FUNCTION "FC_SimNoria" : Void
{ S7_Optimized_Access := 'TRUE' }
VERSION : 2.2
// ==============================================================================
// FC_SimNoria - Симулятор фізики та несправностей норії
// ==============================================================================
// Версія: 2.2.0
// Дата: 2026-04-10
// ==============================================================================
// Зміни v2.2:
//   - Видалено симуляцію DI_Feedback_OK та SimFault_Feedback
//   - Видалено параметри SimFault_Feedback та FaultTime_Feedback_ms
//   - Оновлено симуляцію Noria для Breaker/Alignment
//   - Видалено Feedback_Tripped із внутрішнього стану
// ==============================================================================
// Комунікація з FC_Noria ТІЛЬКИ через сигнали:
//   - Читає:  DB_Mechs.Noria[NoriaIdx].DO_Run
//   - Пише:   DB_Mechs.Noria[NoriaIdx].DI_Speed_OK
//             DB_Mechs.Noria[NoriaIdx].DI_Breaker_OK
//             DB_Mechs.Noria[NoriaIdx].DI_Alingment_OK
// ==============================================================================
   VAR_INPUT
      NoriaIdx : Int;
      StartupTime_ms : DInt;
      StopTime_ms : DInt;
      SimFault_Breaker : Bool;
      FaultTime_Breaker_ms : DInt;
      SimFault_Alignment : Bool;
      FaultTime_Alignment_ms : DInt;
      ManualReset : Bool;
   END_VAR

   VAR_TEMP
      idx : Int;
      elapsedMs : DInt;
      nowTck : DInt;
      startupTimeout : Bool;
      stopTimeout : Bool;
      breakerTimeout : Bool;
      alignmentTimeout : Bool;
   END_VAR


BEGIN
    // =========================================================
    // VALIDATE INDEX
    // =========================================================
    IF #NoriaIdx >= 32 THEN
        RETURN;
    END_IF;

    #idx := #NoriaIdx;

    // =========================================================
    // PHASE 0: Ручний скид аварій
    // =========================================================
    IF #ManualReset THEN
        "DB_SimMechs".Noria[#idx].Breaker_Tripped := FALSE;
        "DB_SimMechs".Noria[#idx].Alignment_Tripped := FALSE;
    END_IF;

    // =========================================================
    // PHASE 1: Edge detection DO_Run
    // =========================================================
    IF "DB_Mechs".Noria[#idx].DO_Run AND NOT "DB_SimMechs".Noria[#idx].LastDO_Run THEN
        "DB_SimMechs".Noria[#idx].MotorStartTck := TIME_TCK();
        "DB_SimMechs".Noria[#idx].FaultStartTck := TIME_TCK();
        "DB_SimMechs".Noria[#idx].IsMotorRunning := TRUE;
        "DB_SimMechs".Noria[#idx].IsSpinningUp := TRUE;
        "DB_SimMechs".Noria[#idx].IsSpinningDown := FALSE;
    END_IF;

    IF NOT "DB_Mechs".Noria[#idx].DO_Run AND "DB_SimMechs".Noria[#idx].LastDO_Run THEN
        "DB_SimMechs".Noria[#idx].MotorStopTck := TIME_TCK();
        "DB_SimMechs".Noria[#idx].IsMotorRunning := FALSE;
        "DB_SimMechs".Noria[#idx].IsSpinningUp := FALSE;
        "DB_SimMechs".Noria[#idx].IsSpinningDown := TRUE;
    END_IF;

    "DB_SimMechs".Noria[#idx].LastDO_Run := "DB_Mechs".Noria[#idx].DO_Run;

    // =========================================================
    // PHASE 2: Симуляція DI_Speed_OK (тахо)
    // =========================================================
    IF "DB_SimMechs".Noria[#idx].IsSpinningUp THEN
        #startupTimeout := "FC_TimeElapsedMs"(
                                              StartTck := "DB_SimMechs".Noria[#idx].MotorStartTck,
                                              TimeoutMs := #StartupTime_ms,
                                              ElapsedMs => #elapsedMs,
                                              NowTck => #nowTck
        );
        IF #startupTimeout THEN
            "DB_Mechs".Noria[#idx].DI_Speed_OK := TRUE;
            "DB_SimMechs".Noria[#idx].IsSpinningUp := FALSE;
        ELSE
            "DB_Mechs".Noria[#idx].DI_Speed_OK := FALSE;
        END_IF;
    ELSIF "DB_SimMechs".Noria[#idx].IsSpinningDown THEN
        #stopTimeout := "FC_TimeElapsedMs"(
                                           StartTck := "DB_SimMechs".Noria[#idx].MotorStopTck,
                                           TimeoutMs := #StopTime_ms,
                                           ElapsedMs => #elapsedMs,
                                           NowTck => #nowTck
        );
        IF #stopTimeout THEN
            "DB_Mechs".Noria[#idx].DI_Speed_OK := FALSE;
            "DB_SimMechs".Noria[#idx].IsSpinningDown := FALSE;
        ELSE
            "DB_Mechs".Noria[#idx].DI_Speed_OK := TRUE;
        END_IF;
    ELSIF "DB_SimMechs".Noria[#idx].IsMotorRunning THEN
        "DB_Mechs".Noria[#idx].DI_Speed_OK := TRUE;
    ELSE
        "DB_Mechs".Noria[#idx].DI_Speed_OK := FALSE;
    END_IF;

    // =========================================================
    // PHASE 4: Симуляція аварії BREAKER
    // =========================================================
    IF #SimFault_Breaker AND "DB_SimMechs".Noria[#idx].IsMotorRunning AND NOT "DB_SimMechs".Noria[#idx].Breaker_Tripped THEN
        #breakerTimeout := "FC_TimeElapsedMs"(
                                              StartTck := "DB_SimMechs".Noria[#idx].FaultStartTck,
                                              TimeoutMs := #FaultTime_Breaker_ms,
                                              ElapsedMs => #elapsedMs,
                                              NowTck => #nowTck
        );
        IF #breakerTimeout THEN
            "DB_SimMechs".Noria[#idx].Breaker_Tripped := TRUE;
        END_IF;
    END_IF;
    "DB_Mechs".Noria[#idx].DI_Breaker_OK := NOT "DB_SimMechs".Noria[#idx].Breaker_Tripped;

    // =========================================================
    // PHASE 5: Симуляція аварії ALIGNMENT
    // =========================================================
    IF #SimFault_Alignment AND "DB_SimMechs".Noria[#idx].IsMotorRunning AND NOT "DB_SimMechs".Noria[#idx].Alignment_Tripped THEN
        #alignmentTimeout := "FC_TimeElapsedMs"(
                                                StartTck := "DB_SimMechs".Noria[#idx].FaultStartTck,
                                                TimeoutMs := #FaultTime_Alignment_ms,
                                                ElapsedMs => #elapsedMs,
                                                NowTck => #nowTck
        );
        IF #alignmentTimeout THEN
            "DB_SimMechs".Noria[#idx].Alignment_Tripped := TRUE;
        END_IF;
    END_IF;
    "DB_Mechs".Noria[#idx].DI_Alingment_OK := NOT "DB_SimMechs".Noria[#idx].Alignment_Tripped;
END_FUNCTION

